// TwinCAT 3 PLC project Untitled1
// ProgramVersion: 3.1.4018.58
// libraries:
//   VisuElem3DPath, 3.5.6.0 (System)
//   VisuElemMeter, 3.5.6.0 (System)
//   VisuElems, 3.5.6.10 (System)
//   VisuElemsDateTime, 3.5.6.0 (System)
//   VisuElemsSpecialControls, 3.5.6.0 (System)
//   VisuElemsWinControls, 3.5.6.0 (System)
//   VisuElemTextEditor, 3.5.6.0 (System)
//   visuinputs, 3.5.6.0 (system)
//   VisuNativeControl, 3.5.6.0 (System)
//   Tc2_Standard, * (Beckhoff Automation GmbH)
//   Tc2_System, * (Beckhoff Automation GmbH)
//   Tc3_Module, * (Beckhoff Automation GmbH)
// project tree:
//   / GlobalTextList.TcGTLO, PlcTask.TcTTO, Visualization Manager.TcVMO (not stored)
//   POUs/ MAIN.TcPOU
//   TxtLst/ Colors.TcTLO
//   VISUs/ VisuAmpel.TcVIS
// real-time tasks:
//   TASK PlcTask: cycle T#10ms, priority 20, ADS port 350

CONFIGURATION Untitled1
    RESOURCE PLC ON TwinCAT3
        TASK PlcTask(INTERVAL := T#10ms, PRIORITY := 20);
        PROGRAM MAIN WITH PlcTask : MAIN;
    END_RESOURCE
END_CONFIGURATION

// ---- POUs/MAIN.TcPOU
PROGRAM MAIN
VAR
	bLight:BOOL; //light enable
	bLightR:BOOL; //turn on R
	bLightG:BOOL; //turn on G
	bLightB:BOOL; //turn on B
	btnSwitch:BOOL; //button signal
	iCounter:DINT; //non persistent turn on counter
	fbTrig:R_TRIG;
	btnText:STRING := 'On'; //text on the toggle button
	iColor:INT:=1; //color choosed
	iWidth:REAL; //line width 
	btnVar:bool; //not used
END_VAR

VAR PERSISTENT  
	iCounterP:DINT; //persistent turn on counter
	iIntensity:REAL; //slider value
END_VAR

fbTrig(CLK:=btnSwitch);


IF fbTrig.Q THEN
	bLight:=NOT bLight;
	IF bLight THEN
		iCounter:=iCOunter+1;
		iCounterP:=iCounterP+1;
	END_IF
END_IF

IF bLight THEN
	CASE iColor OF
		1:
		bLightR:=TRUE;
		bLightG:=FALSE;
		bLightB:=FALSE;
		
		2:
		bLightR:=FALSE;
		bLightG:=TRUE;
		bLightB:=FALSE;
		
		3:
		bLightR:=FALSE;
		bLightG:=FALSE;
		bLightB:=TRUE;
		
		ELSE
		bLightR:=FALSE;
		bLightG:=FALSE;
		bLightB:=FALSE;			
	END_CASE
	btnText:='Off';
	iWidth:=iIntensity;
ELSE
	//turn of the 3 lights
	bLightR:=FALSE;
	bLightG:=FALSE;
	bLightB:=FALSE;	
	btnText:='On';
	iWidth:=0;
END_IF

END_PROGRAM

// ---- GlobalTextList.TcGTLO
TEXTLIST GlobalTextList
  1 = '%s'
  3 = 'Color'
  4 = 'Line width'
  2 = 'NonPersistent: %d'
  0 = 'Persistent: %d'
END_TEXTLIST

// ---- TxtLst/Colors.TcTLO
TEXTLIST Colors
  1 = '1'
  2 = '2'
  3 = '3'
   = ''
END_TEXTLIST

// ---- VISUs/VisuAmpel.TcVIS
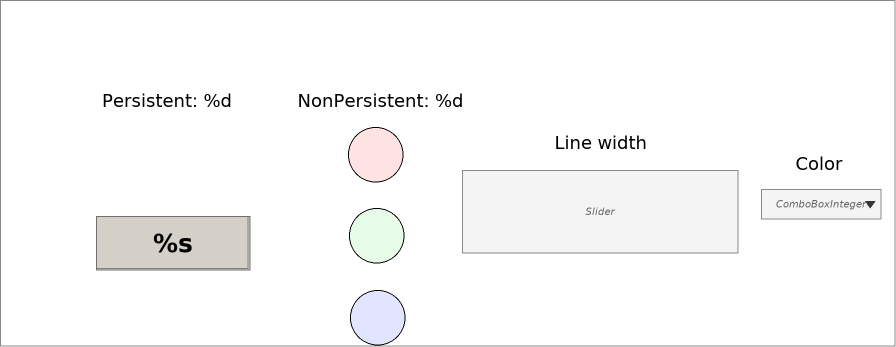
VISUALIZATION VisuAmpel  // 896x347
    Button (96,216 154x54), "%s", text variable: MAIN.btnText
        OnMouseDown: execute { MAIN.btnSwitch:=true; }
        OnMouseUp: execute { MAIN.btnSwitch:=FALSE; }
    Ellipse (348,127 55x55), colour toggle: MAIN.bLightR
        p1271844420: MAIN.iWidth
    Slider (462,170 276x83), variable: MAIN.iIntensity, invisible if: not MAIN.bLight, scale 0..8
    Rectangle (62,78 210x46), "Persistent: %d", text variable: MAIN.iCounterP
    Rectangle (273,78 215x46), "NonPersistent: %d", text variable: MAIN.iCounter
    Ellipse (349,208 55x55), colour toggle: MAIN.bLightG
        p1271844420: MAIN.iWidth
    Ellipse (350,290 55x55), colour toggle: MAIN.bLightB
        p1271844420: MAIN.iWidth
    ComboBoxInteger (761,189 120x30), tooltip "Color", variable: MAIN.iColor, invisible if: not MAIN.bLight, text list: 'Colors'
    Label (526,128 150x30), "Line width", invisible if: not MAIN.bLight
    Label (744,149 150x30), "Color", invisible if: not MAIN.bLight
END_VISUALIZATION
